(* CODESYS project SeasightSolution.library
   Title: Default
   Company: Seasight Solutions
   Version: 1.0.0
   Placeholder: Default

Project tree, tasks and I/O mapping:
  libraries: Tc2_Standard, * (Beckhoff Automation GmbH)
  Components/
    Delta MS300/
      data type E_Delta_MS300_OperationMode
      function block FB_Delta_MS300 [ST]: A_ControlWord, A_Run, A_StateMachine, A_StatusWord
      data type ST_Delta_MS300_ControlWord
      data type ST_Delta_MS300_Input
      data type ST_Delta_MS300_Output
      data type ST_Delta_MS300_StatusWord
  Utils/
    function block FB_LinTrafo [ST]
    function block FB_PulseTrain [ST]
*)

// Components/Delta MS300/E_Delta_MS300_OperationMode
{attribute 'qualified_only'}
{attribute 'strict'}
TYPE E_Delta_MS300_OperationMode :
(
	Reserve,
	ProfilePosition,
	Velocity,
	Reserve2,
	ProfileTorque,
	Reserve3,
	Homing,
	InterpolatedPosition,
	CycliSynchPosition,
	CycliSynchTorque
)SINT;
END_TYPE

// Components/Delta MS300/ST_Delta_MS300_ControlWord
TYPE ST_Delta_MS300_ControlWord :
STRUCT
	SwitchOn: BOOL;
	EnableVoltage: BOOL;
	QuickStop: BOOL;
	EnableOperation: BOOL;
	OperationModeSpecific4: BOOL;
	OperationModeSpecific5: BOOL;
	OperationModeSpecific6: BOOL;
	FaultReset: BOOL;
	Halt: BOOL;
END_STRUCT
END_TYPE

// Components/Delta MS300/ST_Delta_MS300_Input
TYPE ST_Delta_MS300_Input :
STRUCT
	Enable: BOOL;
	Reset: BOOL; // Reset Error/Alarm
	Start: BOOL; // TRUE: Motor ramps to and maintain target velocity. FALSE: Motor ramps to stop.
	
	Velocity: REAL; // [rpm]. Positve => Direction = L1, L2, L3. Negative => Direction = L3, L2, L1.
	GearRatio: REAL; // E.g. 22:7 = 3.14
	
	RampUpTime: REAL; // [s]
	RampDownTime: REAL; // [s]
END_STRUCT
END_TYPE

// Components/Delta MS300/ST_Delta_MS300_Output
TYPE ST_Delta_MS300_Output :
STRUCT
	Fault: BOOL;
	Warning: BOOL;
	ReadyToRun: BOOL;
	TargetReached: BOOL;
	Running: BOOL;
	Ramping: BOOL;
	RampingUp: BOOL;
	RampingDown: BOOL;
	
	ActualVelocity: REAL; // [rpm]
	ActualCurrent: REAL; // [A]
	ActualPower: REAL; // [kW]
END_STRUCT
END_TYPE

// Components/Delta MS300/ST_Delta_MS300_StatusWord
TYPE ST_Delta_MS300_StatusWord :
STRUCT
	ReadyToSwitchOn: BOOL;
	SwitchOn: BOOL;
	OperationEnable: BOOL;
	Fault: BOOL;
	VoltageEnable: BOOL;
	QuickStop: BOOL;
	SwitchOnEnable: BOOL;
	Warning: BOOL;
	Reserved: BOOL;
	Remote: BOOL;
	TargetReached: BOOL;
END_STRUCT
END_TYPE

// Components/Delta MS300/FB_Delta_MS300
FUNCTION_BLOCK FB_Delta_MS300
VAR_INPUT
	stInput: ST_Delta_MS300_Input;
END_VAR
VAR_OUTPUT
	stOutput: ST_Delta_MS300_Output;
END_VAR
VAR
	stStat: ST_Delta_MS300_StatusWord;
	stCtrl: ST_Delta_MS300_ControlWord;
	
	nStatusWord AT %I*: UINT;
	nActualVelocity AT %I*: UINT; // [rpm]
	nActualCurrent AT %I*: UINT; // [1/100 A]
	nActualPower AT %I*: UINT; // [1/10 kW]
	nModeOperationStat AT %I*: SINT;
	
	nControlWord AT %Q*: UINT;
	nTargetVelocity AT %Q*: INT; // [rpm]
	nModeOperationCtrl AT %Q*: SINT;
	
	nRampUpTime AT %Q*: UDINT; // [ms]
	nRampDownTime AT %Q*: UDINT; // [ms]
	
	nState: INT;
	tonResetTimeout: TON;
END_VAR

A_Run();

A_StatusWord();
A_ControlWord();

A_StateMachine();

ACTION A_ControlWord:
nControlWord.0 := stCtrl.SwitchOn;
nControlWord.1 := stCtrl.EnableVoltage;
nControlWord.2 := stCtrl.QuickStop;
nControlWord.3 := stCtrl.EnableOperation;
nControlWord.4 := stCtrl.OperationModeSpecific4;
nControlWord.5 := stCtrl.OperationModeSpecific5;
nControlWord.6 := stCtrl.OperationModeSpecific6;
nControlWord.7 := stCtrl.FaultReset;
nControlWord.8 := stCtrl.Halt;
END_ACTION

ACTION A_Run:
//////////////////////////////
//			Input			//
//////////////////////////////

// Set Operation Mode
nModeOperationCtrl := E_Delta_MS300_OperationMode.Velocity;

// Set ramp time
nRampUpTime := TO_UDINT(stInput.RampUpTime * 1E3);
nRampDownTime := TO_UDINT(stInput.RampDownTime * 1E3);

//Set target velocity
nTargetVelocity := TO_INT(stInput.Velocity * stInput.GearRatio);

// Start signals
// Maintain current speed; B4 and B6.
// Run to target speed: B4, B5, and B6.
// Decelerate to 0 rpm: None
stCtrl.OperationModeSpecific4 := stInput.Start;
stCtrl.OperationModeSpecific5 := stInput.Start;
stCtrl.OperationModeSpecific6 := stInput.Start;

//////////////////////////////
//			Output			//
//////////////////////////////

// Target speed reached
stOutput.TargetReached := stStat.TargetReached;

// Ramping
stOutput.Ramping := stOutput.ActualVelocity > 10 AND NOT stOutput.TargetReached;

// Ramping up
stOutput.RampingUp := stInput.Start AND stOutput.ActualVelocity > 10 AND NOT stOutput.TargetReached;

// Ramping down
stOutput.RampingDown := NOT stInput.Start AND stOutput.ActualVelocity > 10;

// Running
stOutput.Running := stOutput.ActualVelocity > 10;

// Actual current
stOutput.ActualCurrent := TO_REAL(nActualCurrent) / 100;

// Actual power
stOutput.ActualPower := TO_REAL(nActualPower) / 10;

// Actual Velocity
IF stInput.GearRatio > 0 THEN
	stOutput.ActualVelocity := TO_REAL(nActualVelocity) / stInput.GearRatio;
ELSE
	stOutput.ActualVelocity := TO_REAL(nActualVelocity);
END_IF
END_ACTION

ACTION A_StateMachine:
stCtrl.SwitchOn := FALSE;
stCtrl.EnableVoltage := FALSE;
stCtrl.QuickStop := FALSE;
stCtrl.EnableOperation := FALSE;
stCtrl.OperationModeSpecific4 := FALSE;
stCtrl.OperationModeSpecific5 := FALSE;
stCtrl.OperationModeSpecific6 := FALSE;
stCtrl.Halt := FALSE;

stOutput.ReadyToRun := FALSE;

IF NOT stInput.Enable THEN
	nState := 0;
END_IF

CASE nState OF
	0:	// Not ready to switch on
		IF stStat.SwitchOnEnable AND stInput.Enable THEN
			nState := nState + 1;
		END_IF
		
	1:	// Switch on disabled
		stCtrl.EnableVoltage := TRUE;
		stCtrl.QuickStop := TRUE;
		IF stStat.ReadyToSwitchOn AND stStat.QuickStop THEN
			nState := nState + 1;
		END_IF
		
	2:	// Ready to switch on
		stCtrl.SwitchOn := TRUE;
		stCtrl.EnableVoltage := TRUE;
		stCtrl.QuickStop := TRUE;
		IF stStat.ReadyToSwitchOn AND stStat.SwitchOn AND stStat.QuickStop THEN
			nState := nState + 1;
		END_IF
		
	3:	// Switch on
		stCtrl.SwitchOn := TRUE;
		stCtrl.EnableVoltage := TRUE;
		stCtrl.QuickStop := TRUE;
		stCtrl.EnableOperation := TRUE;
		IF stStat.ReadyToSwitchOn AND stStat.SwitchOn AND stStat.OperationEnable AND stStat.QuickStop THEN
			nState := nState + 1;
		END_IF
		
	4:	// Operation enabled
		stCtrl.SwitchOn := TRUE;
		stCtrl.EnableVoltage := TRUE;
		stCtrl.QuickStop := TRUE;
		stCtrl.EnableOperation := TRUE;
		
		stOutput.ReadyToRun := TRUE;
		
		IF NOT stStat.ReadyToSwitchOn OR NOT stStat.SwitchOn OR NOT stStat.OperationEnable OR NOT stStat.QuickStop THEN
			nState := 1;
		END_IF
END_CASE
END_ACTION

ACTION A_StatusWord:
stStat.ReadyToSwitchOn := nStatusWord.0;
stStat.SwitchOn := nStatusWord.1;
stStat.OperationEnable := nStatusWord.2;
stStat.Fault := nStatusWord.3;
stStat.VoltageEnable := nStatusWord.4;
stStat.QuickStop := nStatusWord.5;
stStat.SwitchOnEnable := nStatusWord.6;
stStat.Warning := nStatusWord.7;
stStat.Reserved := nStatusWord.8;
stStat.Remote := nStatusWord.9;
stStat.TargetReached := nStatusWord.10;
END_ACTION

END_FUNCTION_BLOCK

// Utils/FB_LinTrafo
FUNCTION_BLOCK FB_LinTrafo
VAR_INPUT
	fInputValue: LREAL;
	fInMin: LREAL;
	fInMax: LREAL;
	fOutMin: LREAL;
	fOutMax: LREAL;
END_VAR
VAR_OUTPUT
	fOutputValue: LREAL;
END_VAR
VAR
	fSlope: LREAL;
	fIntersection: LREAL;
END_VAR

IF fInMin - fInMax <> 0.0 THEN
	fSlope := (fOutMax - fOutMin) / (fInMax - fInMin);
	fIntersection := fOutMax - fSlope * fInMax;
	fOutputValue := fInputValue * fSlope + fIntersection;
END_IF

END_FUNCTION_BLOCK

// Utils/FB_PulseTrain
FUNCTION_BLOCK FB_PulseTrain
VAR_INPUT
	bStart: BOOL;
	
	tPulseOn: TIME := T#200MS;
	tPulseOff: TIME := T#200MS;
END_VAR
VAR_OUTPUT
	bPulse: BOOL;
	bOnePulse: BOOL;
END_VAR
VAR
	rtOnePulse: R_TRIG;
	tonPulseOn: TON := (PT := tPulseOn);
	tonPulseOff: TON := (PT := tPulseOff);
END_VAR

// One-Pulse-Trigger
rtOnePulse(CLK := bStart, Q => bOnePulse);

// bPulse always starts TRUE
IF bOnePulse THEN bPulse := TRUE; END_IF
	tonPulseOn(IN := bPulse);
	tonPulseOff(IN := NOT bPulse);
IF bStart AND tonPulseOn.Q THEN
	bPulse := FALSE;
ELSIF bStart AND tonPulseOff.Q THEN
	bPulse := TRUE;
END_IF

END_FUNCTION_BLOCK
